// TIA Portal V16 export
// export: Created 2022-02-11T10:45:12.248232Z, ExportSetting WithDefaults, DisplayName Totally Integrated Automation Portal, DisplayVersion V16 Update 5, DisplayName TIA Portal Version Control Interface, DisplayVersion V16 Update 2, DisplayName TIA Portal Openness, DisplayVersion V16 Update 5, DisplayName STEP 7 Professional, DisplayVersion V16 Update 5, DisplayName STEP 7 Safety, DisplayVersion V16, DisplayName WinCC Professional, DisplayVersion V16 Update 5, DisplayName SIMATIC Visualization Architect, DisplayVersion V16
FUNCTION_BLOCK "fbObjEV_Mono_NC_AmbDP"   // FB9101, LAD
{ S7_Optimized_Access := 'TRUE' }
VERSION : 0.1
// stored: AutoNumber false, IsIECCheckEnabled false, IsRetainMemResEnabled false, MemoryReserve 0, SetENOAutomatically false, UDAEnableTagReadback false
   VAR_INPUT
      eDP_Oberta : Bool := FALSE;   // Detector posicio valvula oberta
      eDP_Tancada : Bool := TRUE;   // Detector posicio valvula tancada
      aOpenAuto : Bool := FALSE;   // Ordre obrir EV en automatic
      psEnaAutoGrl : "boto";
      psEnaManualGrl : "boto";
      bCM_Open : Bool := TRUE;   // Condicions necesaries obrir valvula
      tAla_Open : Time := t#5s;   // Temps retard activacio alarma error obrir EV
      tAla_Close : Time := t#5s;   // Temps retard activacio alarma error tancar EV
      tAla_CM_Open : Time := t#3s;   // Temps retard activacio alarma condicions moviment
      psAnuConMov : Bool;
      psResetAlarma : Bool;
      mFirstScan : Bool;
      "Clock_0.5Hz" : Bool;
      bSysOk : Bool;
   END_VAR
   VAR_OUTPUT
      aOpen : Bool;   // Sortida activacio EV
      be_Open : Bool;   // Bit estat EV oberta (Detectors + Sortida)
      be_Close : Bool;   // Bit estat EV tancada (Detectors + Sortida)
      al_CM_Open : Bool;   // Alarma condicions moviment obrir
      al_Open : Bool;   // Alarma obrir EV
      al_Close : Bool;   // Alarma tancar EV
      al_psEna : Bool;
   END_VAR
   VAR
      HMI : "HMI_oEV";
      timAla_CM_Open : IEC_TIMER;   // Timer retard alarma condicions moviment
      timAla_Open : IEC_TIMER;   // Timer retard alarma obrirEV
      timAla_Close : IEC_TIMER;   // Timer retard alarma tancar EV
      mAuxTimer : Bool;   // Bit auxiliarInicialitzacio timers
      bLast_Reset : Bool;
   END_VAR
   VAR_TEMP
      _ModeAutomatic : Bool;
      _ModeManual : Bool;
      be_Open_Err : Bool;   // Error en validacio EV oberta. Sense retard per alarma.
      be_Close_Err : Bool;   // Error en validacio EV tancada. Sense retard per alarma.
      bErrorCM : Bool;   // Error CM. Si activem sortida i no es compleixen les CM. Sense retard
      aOpenSenseTestCM : Bool;
      bCM_Ok : Bool;
      ResetAlarmes : Bool;
   END_VAR
   VAR CONSTANT
      STATUS_OBJ_ERR : Int := 10;
      STATUS_OBJ_WARNING : Int := 11;
      STATUS_OBJ_ON : Int := 1;
      STATUS_OBJ_OFF : Int := 0;
      STATUS_OBJ_UNKNOWN : Int := -1;
   END_VAR
   VAR_TEMP   // added for the SCL form of the ladder/FBD networks
      _w1 : Bool;
   END_VAR
BEGIN

REGION Network 1 (SCL): Descripció
   // Motor activat per Rele, amb confirmacio i proteccio.
END_REGION

REGION Network 2: Test habilitació mode manual. Desactivar si no tenim polsador manual o no tenim maniobra.
   // psEnaManualGrl : és el pulsador de manual de Appinfo. Si aquest està activar tots els objectes del cicle es troben en Mode Manual.
   // 
   // HMI.psEnaManual : és el pulsador de manual únic de l'objecte. Significa que la resta d'objectes es trobaràn en automàtic menys aquest.
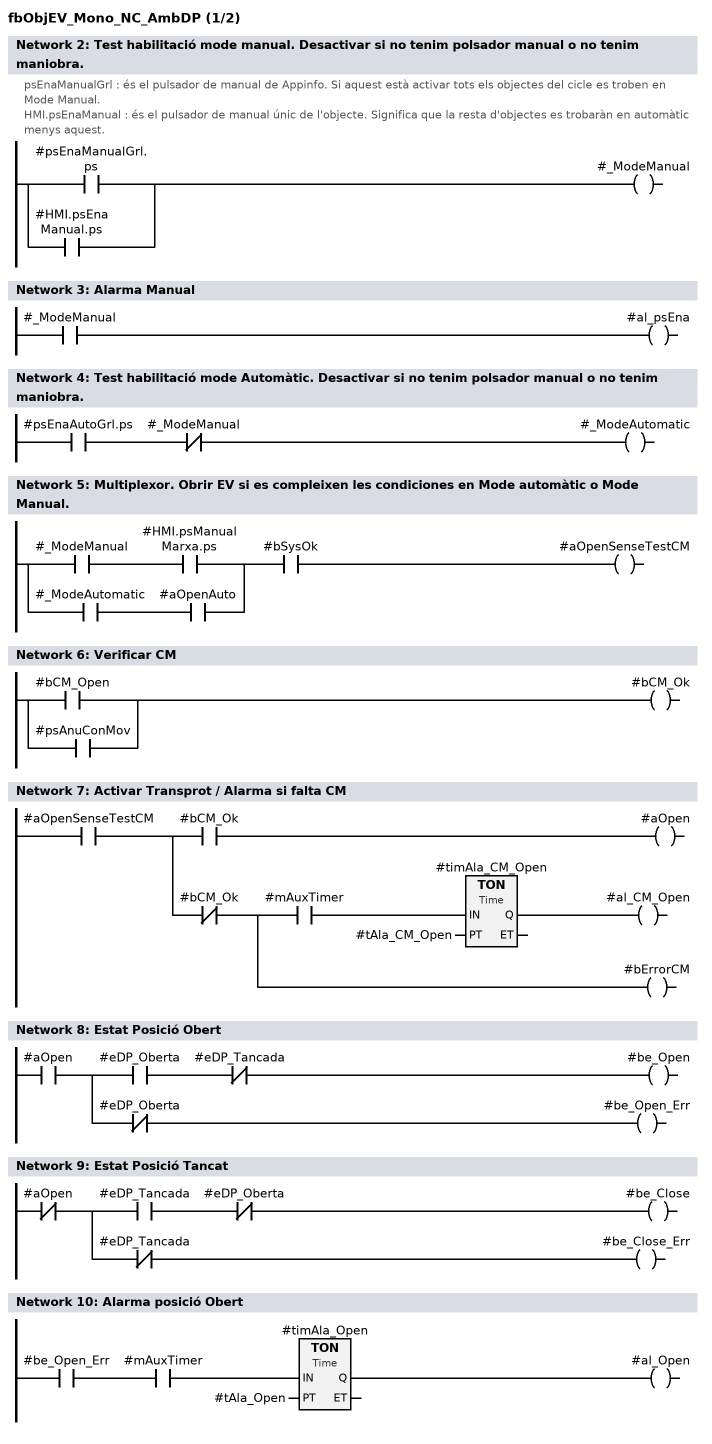
   RUNG wire#powerrail
      Contact( #psEnaManualGrl.ps )
      wire#w1
      Coil( #_ModeManual )
   END_RUNG
   RUNG wire#powerrail
      Contact( #HMI.psEnaManual.ps )
   END_RUNG wire#w1
   // the same network as SCL:
   #_ModeManual := #psEnaManualGrl.ps OR #HMI.psEnaManual.ps;
END_REGION

REGION Network 3: Alarma Manual
   RUNG wire#powerrail
      Contact( #_ModeManual )
      Coil( #al_psEna )
   END_RUNG
   // the same network as SCL:
   #al_psEna := #_ModeManual;
END_REGION

REGION Network 4: Test habilitació mode Automàtic. Desactivar si no tenim polsador manual o no tenim maniobra.
   RUNG wire#powerrail
      Contact( #psEnaAutoGrl.ps )
      I_Contact( #_ModeManual )
      Coil( #_ModeAutomatic )
   END_RUNG
   // the same network as SCL:
   #_ModeAutomatic := #psEnaAutoGrl.ps AND NOT #_ModeManual;
END_REGION

REGION Network 5: Multiplexor. Obrir EV si es compleixen les condiciones en Mode automàtic o Mode Manual.
   RUNG wire#powerrail
      Contact( #_ModeManual )
      Contact( #HMI.psManualMarxa.ps )
      wire#w1
      Contact( #bSysOk )
      Coil( #aOpenSenseTestCM )
   END_RUNG
   RUNG wire#powerrail
      Contact( #_ModeAutomatic )
      Contact( #aOpenAuto )
   END_RUNG wire#w1
   // the same network as SCL:
   #aOpenSenseTestCM := ((#_ModeManual AND #HMI.psManualMarxa.ps) OR (#_ModeAutomatic AND #aOpenAuto)) AND #bSysOk;
END_REGION

REGION Network 6: Verificar CM
   RUNG wire#powerrail
      Contact( #bCM_Open )
      wire#w1
      Coil( #bCM_Ok )
   END_RUNG
   RUNG wire#powerrail
      Contact( #psAnuConMov )
   END_RUNG wire#w1
   // the same network as SCL:
   #bCM_Ok := #bCM_Open OR #psAnuConMov;
END_REGION

REGION Network 7: Activar Transprot / Alarma si falta CM
   RUNG wire#powerrail
      Contact( #aOpenSenseTestCM )
      wire#w1
      Contact( #bCM_Ok )
      Coil( #aOpen )
   END_RUNG
   RUNG wire#w1
      I_Contact( #bCM_Ok )
      wire#w2
      Contact( #mAuxTimer )
      { S7_Templates := "time_type := Time" } #timAla_CM_Open.TON(pt := #tAla_CM_Open, et =>)
      Coil( #al_CM_Open )
   END_RUNG
   RUNG wire#w2
      Coil( #bErrorCM )
   END_RUNG
   // the same network as SCL:
   #aOpen := #aOpenSenseTestCM AND #bCM_Ok;
   #_w1 := #aOpenSenseTestCM AND NOT #bCM_Ok;
   #timAla_CM_Open.TON(IN := #_w1 AND #mAuxTimer, PT := #tAla_CM_Open);
   #al_CM_Open := #timAla_CM_Open.Q;
   #bErrorCM := #_w1;
END_REGION

REGION Network 8: Estat Posició Obert
   RUNG wire#powerrail
      Contact( #aOpen )
      wire#w1
      Contact( #eDP_Oberta )
      I_Contact( #eDP_Tancada )
      Coil( #be_Open )
   END_RUNG
   RUNG wire#w1
      I_Contact( #eDP_Oberta )
      Coil( #be_Open_Err )
   END_RUNG
   // the same network as SCL:
   #be_Open := #aOpen AND #eDP_Oberta AND NOT #eDP_Tancada;
   #be_Open_Err := #aOpen AND NOT #eDP_Oberta;
END_REGION

REGION Network 9: Estat Posició Tancat
   RUNG wire#powerrail
      I_Contact( #aOpen )
      wire#w1
      Contact( #eDP_Tancada )
      I_Contact( #eDP_Oberta )
      Coil( #be_Close )
   END_RUNG
   RUNG wire#w1
      I_Contact( #eDP_Tancada )
      Coil( #be_Close_Err )
   END_RUNG
   // the same network as SCL:
   #be_Close := NOT #aOpen AND #eDP_Tancada AND NOT #eDP_Oberta;
   #be_Close_Err := NOT #aOpen AND NOT #eDP_Tancada;
END_REGION

REGION Network 10: Alarma posició Obert
   RUNG wire#powerrail
      Contact( #be_Open_Err )
      Contact( #mAuxTimer )
      { S7_Templates := "time_type := Time" } #timAla_Open.TON(pt := #tAla_Open, et =>)
      Coil( #al_Open )
   END_RUNG
   // the same network as SCL:
   #timAla_Open.TON(IN := #be_Open_Err AND #mAuxTimer, PT := #tAla_Open);
   #al_Open := #timAla_Open.Q;
END_REGION

REGION Network 11: Alarma posició tancat
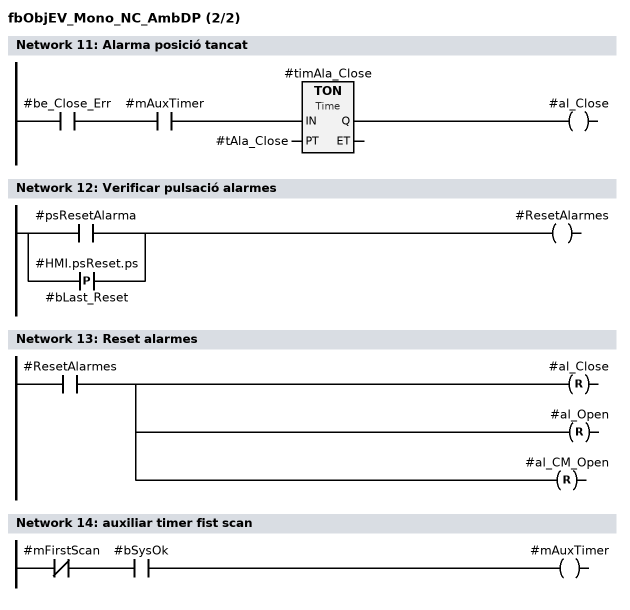
   RUNG wire#powerrail
      Contact( #be_Close_Err )
      Contact( #mAuxTimer )
      { S7_Templates := "time_type := Time" } #timAla_Close.TON(pt := #tAla_Close, et =>)
      Coil( #al_Close )
   END_RUNG
   // the same network as SCL:
   #timAla_Close.TON(IN := #be_Close_Err AND #mAuxTimer, PT := #tAla_Close);
   #al_Close := #timAla_Close.Q;
END_REGION

REGION Network 12: Verificar pulsació alarmes
   RUNG wire#powerrail
      Contact( #psResetAlarma )
      wire#w1
      Coil( #ResetAlarmes )
   END_RUNG
   RUNG wire#powerrail
      P_Contact(operand := #HMI.psReset.ps, bit := #bLast_Reset)
   END_RUNG wire#w1
   // the same network as SCL:
   #_w1 := #HMI.psReset.ps AND NOT #bLast_Reset;   // rising edge of #HMI.psReset.ps
   #bLast_Reset := #HMI.psReset.ps;
   #ResetAlarmes := #psResetAlarma OR #_w1;
END_REGION

REGION Network 13: Reset alarmes
   RUNG wire#powerrail
      Contact( #ResetAlarmes )
      wire#w1
      R_Coil( #al_Close )
   END_RUNG
   RUNG wire#w1
      R_Coil( #al_Open )
   END_RUNG
   RUNG wire#w1
      R_Coil( #al_CM_Open )
   END_RUNG
   // the same network as SCL:
   IF #ResetAlarmes THEN
       #al_Close := FALSE;
       #al_Open := FALSE;
       #al_CM_Open := FALSE;
   END_IF;
END_REGION

REGION Network 14: auxiliar timer fist scan
   RUNG wire#powerrail
      I_Contact( #mFirstScan )
      Contact( #bSysOk )
      Coil( #mAuxTimer )
   END_RUNG
   // the same network as SCL:
   #mAuxTimer := NOT #mFirstScan AND #bSysOk;
END_REGION

REGION Network 15 (SCL): HMI estat EV
       IF (#al_Open OR #al_Close OR #al_CM_Open) THEN
           #HMI.iStatusDisplay := #STATUS_OBJ_ERR;                // Error = 10
           #HMI.bDisplayError := TRUE;
           #HMI.bDisplayWarning := FALSE;
           #HMI.bDisplayOk := FALSE;

       ELSIF (#be_Open_Err OR #be_Close_Err) THEN
           #HMI.iStatusDisplay := #STATUS_OBJ_WARNING;            // Warning = 11
           #HMI.bDisplayError := FALSE;
           #HMI.bDisplayWarning := TRUE;
           #HMI.bDisplayOk := FALSE;

       ELSIF #be_Open THEN
           #HMI.iStatusDisplay := #STATUS_OBJ_ON;                 // Bit estat Open Auto = 1
           #HMI.bDisplayError := FALSE;
           #HMI.bDisplayWarning := FALSE;
           #HMI.bDisplayOk := TRUE;

       ELSIF #be_Close THEN
           #HMI.iStatusDisplay := #STATUS_OBJ_OFF;               // Bit estat Close Automatic = 0
           #HMI.bDisplayError := FALSE;
           #HMI.bDisplayWarning := FALSE;
           #HMI.bDisplayOk := TRUE;

       ELSIF #aOpen THEN
           IF #"Clock_0.5Hz" THEN
               #HMI.iStatusDisplay := #STATUS_OBJ_ON;
           ELSE
               #HMI.iStatusDisplay := #STATUS_OBJ_WARNING;
           END_IF;
           #HMI.bDisplayError := FALSE;
           #HMI.bDisplayWarning := FALSE;
           #HMI.bDisplayOk := TRUE;

       ELSE
           #HMI.iStatusDisplay := #STATUS_OBJ_UNKNOWN;            // Unknown = -1
           #HMI.bDisplayError := TRUE;
           #HMI.bDisplayWarning := FALSE;
           #HMI.bDisplayOk := FALSE;

       END_IF;

       #HMI.eON := #aOpen;
       #HMI.eOFF := NOT #aOpen;
       #HMI.error := #al_CM_Open OR #al_Open OR #al_Close;
       #HMI.confirmacio := #bSysOk;
END_REGION
END_FUNCTION_BLOCK
